// TIA Portal project "Automatisierte Nussfüllstation_SCL" (V16)

(* hardware
DEVICE "S7-1200 station_1"  S7-1200 Station
   slot 0: "Rack_0"  S7-1200 Rack  Rack  V1.0
   slot 1: "PLC_1"  CPU 1212C DC/DC/DC  6ES7 212-1AE40-0XB0  V4.4
*)

// ===== PLC "PLC_1"  CPU 1212C DC/DC/DC =====

VAR_GLOBAL   // PLC tag table "Default tag table"
   "Eingang_Näherungssensor" AT %I0.0 : Bool;
   "Eingang_Ultraschallfüllstandsensor" AT %I0.1 : Bool;
   "Kontaktstelle Farbsensor (ROT)" AT %I0.2 : Bool;
   "Kontaktstelle Farbsensor (BLAU)" AT %I0.3 : Bool;
   "Ausgang_Motor" AT %Q0.0 : Bool;
   "Ausgang_Walnusszufuhrklappe" AT %Q0.1 : Bool;
   "Ausgang_Pekanzufuhrklappe" AT %Q0.2 : Bool;
   "Näherungssensor_Bit" AT %M0.0 : Bool;
   "Ultraschallfüllstandsensor_Bit" AT %M0.1 : Bool;
   "Farbsensor_ROT_Bit" AT %M0.3 : Bool;
   "Farbsensor_BLAU_Bit" AT %M0.4 : Bool;
   "Motor_Bit" AT %M0.5 : Bool;
   "Walnusszufuhrklappe_Bit" AT %M0.6 : Bool;
   "Pekanzufuhrklappe_Bit" AT %M0.7 : Bool;
   "Modus" AT %MW2 : Int;
END_VAR

DATA_BLOCK "IO_DB"   // DB1
{ S7_Optimized_Access := 'TRUE' }
VERSION : 0.1
// stored: InstanceOfName IO
"IO"
BEGIN
END_DATA_BLOCK

DATA_BLOCK "Steuerlogik_DB"   // DB2
{ S7_Optimized_Access := 'TRUE' }
VERSION : 0.1
// stored: InstanceOfName Steuerlogik
"Steuerlogik"
BEGIN
END_DATA_BLOCK

FUNCTION_BLOCK "IO"   // FB1, SCL
{ S7_Optimized_Access := 'TRUE' }
VERSION : 0.1
BEGIN
   // Eingänge
       IF "Eingang_Näherungssensor" THEN
           "Näherungssensor_Bit" := TRUE;
       ELSE
           "Näherungssensor_Bit" := FALSE;
       END_IF;

       IF "Eingang_Ultraschallfüllstandsensor" THEN
           "Ultraschallfüllstandsensor_Bit" := TRUE;
       ELSE
           "Ultraschallfüllstandsensor_Bit" := FALSE;
       END_IF;

       IF "Kontaktstelle Farbsensor (ROT)" THEN
           "Farbsensor_ROT_Bit" := TRUE;
       ELSE
           "Farbsensor_ROT_Bit" := FALSE;
       END_IF;

       IF "Kontaktstelle Farbsensor (BLAU)" THEN
           "Farbsensor_BLAU_Bit" := TRUE;
       ELSE
           "Farbsensor_BLAU_Bit" := FALSE;
       END_IF;


   // Ausgänge
       IF "Motor_Bit" THEN
           "Ausgang_Motor" := TRUE;
       ELSE
           "Ausgang_Motor" := FALSE;
   END_IF;

   IF "Walnusszufuhrklappe_Bit" THEN
       "Ausgang_Walnusszufuhrklappe" := TRUE;
   ELSE
       "Ausgang_Walnusszufuhrklappe" := FALSE;
   END_IF;

   IF "Pekanzufuhrklappe_Bit" THEN
       "Ausgang_Pekanzufuhrklappe" := TRUE;
   ELSE
       "Ausgang_Pekanzufuhrklappe" := FALSE;
   END_IF;
END_FUNCTION_BLOCK

FUNCTION_BLOCK "Steuerlogik"   // FB2, SCL
{ S7_Optimized_Access := 'TRUE' }
VERSION : 0.1
BEGIN
   IF NOT "Näherungssensor_Bit" AND NOT "Ultraschallfüllstandsensor_Bit" AND NOT "Farbsensor_ROT_Bit" AND NOT "Farbsensor_BLAU_Bit" THEN
       "Modus" := 1;
   END_IF;
   // Modus:
   // 1 = Motor an;
   // 2 = Füllmodus
   IF "Näherungssensor_Bit" AND NOT "Ultraschallfüllstandsensor_Bit" THEN
       "Modus" := 2;
   END_IF;

   IF "Näherungssensor_Bit" AND "Ultraschallfüllstandsensor_Bit" AND ("Farbsensor_BLAU_Bit" OR "Farbsensor_ROT_Bit") THEN
       "Modus" := 1;
   END_IF;

   IF "Modus" = 1 THEN
       "Motor_Bit" := TRUE;
   ELSE
       "Motor_Bit" := FALSE;
   END_IF;

   IF "Modus" = 2 AND "Farbsensor_ROT_Bit" AND NOT "Farbsensor_BLAU_Bit" AND NOT "Ultraschallfüllstandsensor_Bit" AND "Näherungssensor_Bit" THEN
       "Pekanzufuhrklappe_Bit" := TRUE;
   ELSE
       "Pekanzufuhrklappe_Bit" := FALSE;
   END_IF;

   IF "Modus" = 2 AND "Farbsensor_BLAU_Bit" AND NOT "Farbsensor_ROT_Bit" AND NOT "Ultraschallfüllstandsensor_Bit" AND "Näherungssensor_Bit" THEN
       "Walnusszufuhrklappe_Bit" := TRUE;
   ELSE
       "Walnusszufuhrklappe_Bit" := FALSE;
       END_IF;
END_FUNCTION_BLOCK

ORGANIZATION_BLOCK "Main"   // OB1, LAD, ProgramCycle
TITLE = "Main Program Sweep (Cycle)"
{ S7_Optimized_Access := 'TRUE' }
VERSION : 0.1
// PROJEKTBESCHREIBUNG.: In diesem Projekt geht um die automatische Nussabfüllmaschine. Die Anlage besteht aus einem Motor, einem Förderband, einem Näherungssensor, zwei Nusstrichter (Pekan- und Walnusstrichter) mti Zufuhrklappen, einem Farbsensor (erkennt rot und blau) und einem Ultraschallfüllstandsensor. Die Reihenfolge der Steuerlogik ist wie folgt:
// 1)  Auf dem Förderband liegen die abzufüllenden Kartonverpackungen. Der Motor geht an und somit bewegt den Förderband bis der Näherungssensor die Kartonverpackung erkennt.
// 2) Auf der Kartonverpackung ist jeweils eine rote oder blaue Etikettierung.Der Farbsensor erkennt die Farbe und anhand dieser Farbe (rot für Pekannüsse und blau für Walnüsse) wird jeweiligen Zufuhrklappen zur Befüllung geöffnet.
// 3) Der Ultraschallfüllstandsensor misst ständig ,ob die Verpackung voll ist. Falls ja, die Zufuhrklappe ist geschlossen und der Förderband bewegt die befüllte Verpackung weiter.  
// 
// TESTKRITERIEN:
// 1)Um zu beginnen, starten Sie Ihr Programm auf PLCSIM. Der Fördermotor sollte sofort anlaufen, aber beide Trichter sollten ausgeschaltet sein.
// 
// 2)Als Nächstes erzwingen Sie nur den Näherungsschalter (geschlossen). Der Fördermotor sollte sich abschalten, und beide Trichter sollten ausgeschaltet bleiben.
// 
// 3)Drittens lassen Sie den Näherungsschalter geschlossen und erzwingen zusätzlich die rote Lichtschranke. Der Fördermotor und der Walnuss-Trichter sollten ausgeschaltet bleiben, aber der Pekannuss-Trichter sollte einschalten.
// 
// 4)Viertens lassen Sie den Näherungsschalter geschlossen, schalten die rote Lichtschranke aus und erzwingen die blaue Lichtschranke. Der Fördermotor sollte ausgeschaltet bleiben, der Pekannuss-Trichter sollte ausgehen und der Walnuss-Trichter sollte einschalten.
// 
// 5)Als Nächstes erzwingen Sie den Füllstandsschalter. Beide Trichter sollten ausgeschaltet werden und der Förderer sollte wieder anlaufen, um die Kiste weiterzubewegen.
// 
// 6)Zum Schluss schalten Sie den Näherungsschalter, den Füllstandsschalter und beide Lichtschranken aus. Beide Trichter sollten ausgeschaltet bleiben und der Förderer sollte weiterlaufen.
// 7)
// Zusatztest: Bei geöffnetem Näherungsschalter und Füllstandsschalter erzwingen Sie beide Lichtschranken. Keiner der Trichter sollte einschalten. (Wir wollen kein Produkt freigeben, wenn keine Kiste zum Auffangen da ist.)
   VAR_INPUT
      Initial_Call : Bool;   // Initial call of this OB
      Remanence : Bool;   // =True, if remanent data are available
   END_VAR
BEGIN

REGION Network 1
   // IO
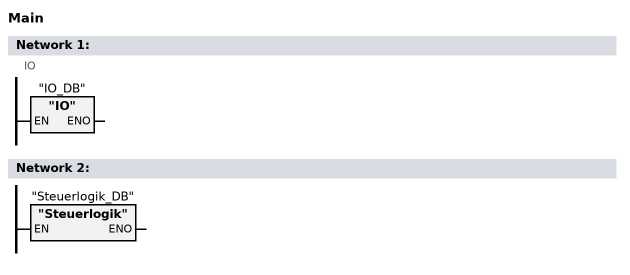
   RUNG wire#powerrail
      "IO_DB"()
   END_RUNG
   // the same network as SCL:
   "IO_DB"();   // "IO"
END_REGION

REGION Network 2
   RUNG wire#powerrail
      "Steuerlogik_DB"()
   END_RUNG
   // the same network as SCL:
   "Steuerlogik_DB"();   // "Steuerlogik"
END_REGION
END_ORGANIZATION_BLOCK